// TIA Portal V20 export
DATA_BLOCK "SP511"   // DB327
// stored: MemoryReserve 100
   VAR
      SPARE : Bool;
      SPARE_1 : Bool;
      SPARE_2 : Bool;
      SPARE_3 : Bool;
      SPARE_4 : Bool;
      SPARE_5 : Bool;
      SPARE_6 : Bool;
      SPARE_7 : Bool;
      SPARE_8 : Bool;
      SPARE_9 : Bool;
      "HEATER-1 TEMPERATURE CONTROLLER RS485" : Bool;
      SPARE_10 : Bool;
      SPARE_11 : Bool;
      SPARE_12 : Bool;
      SPARE_13 : Bool;
      SPARE_14 : Bool;
   END_VAR
BEGIN
END_DATA_BLOCK
